TYPE ST_PermIntlkIndex :
STRUCT
	Condition : BOOL := TRUE;
	Description : STRING(Param_PermIntlk.DESCRIPTION_LEN);
END_STRUCT
END_TYPE

(* stored: Version 1.1.0.1, ProductVersion 3.1.4024.12
   DUT ST_PermIntlkIndex: Id {2024c61a-99cb-4347-9d90-16bbb126dd07} *)
